PROGRAM MAIN
VAR
	Axis		: ARRAY [0..1] OF CNC_Axis; // CNC axis
	Hli 		: MCV_HliInterface;
	axisIdx		: UINT;
END_VAR

(* configuration *)
Axis[0].config.driveId	:= 1001;				// Drive 1 (TSD)/EtherCAT/EtherCAT-Addr.
Axis[0].config.netId	:= '10.20.34.98.2.1';	// Drive 1 (TSD)^InfoData^AdsAddr^netId
Axis[0].config.axisNumber:= 0;					// first (0) or second (1) axis of a dual axis drive
Axis[0].config.axisId	:= 0;					// cnc-axis-id used in events
Axis[1].config.driveId	:= 1001;				// Drive 1 (TSD)/EtherCAT/EtherCAT-Addr.
Axis[1].config.netId	:= '10.20.34.98.2.1';	// Drive 1 (TSD)^InfoData^AdsAddr^netId
Axis[1].config.axisNumber:= 1;					// first (0) or second (1) axis of a dual axis drive
Axis[1].config.axisId	:= 1;					// cnc-axis-id used in events

(* HLI interface *)
IF NOT Hli.Initialized THEN
	Hli(); //initialize HLI
END_IF

(* Axis handler *)
IF Hli.Initialized THEN
	gStatusAxesEnabled := TRUE;
	FOR axisIdx := 0 TO SIZEOF(Axis)/SIZEOF(Axis[0])-1 DO
		Axis[axisIdx].enable := gEnableAxes;
		Axis[axisIdx]();
		IF NOT Axis[axisIdx].enabled THEN
			gStatusAxesEnabled := FALSE;
		END_IF
	END_FOR
END_IF

END_PROGRAM

(* stored: Version 1.1.0.1, ProductVersion 3.1.4024.12
   POU MAIN: Id {99e0d0d8-73f4-4a0e-9efd-bf064104c456}, SpecialFunc None *)
